INTERFACE Evaluable

METHOD evalue : Awaitable
VAR_INPUT
	value: BOOL;
	onTrueCallback: Callback;
	onFalseCallback: REFERENCE TO AwaitableError;
	message: STRING(255);
END_VAR
END_METHOD

END_INTERFACE

(* stored: Version 1.1.0.1, ProductVersion 3.1.4024.12
   Itf Evaluable: Id {5fdc8daf-5053-4b6d-a120-f929bb45a04c}
   Method evalue: Id {ba9f3a6b-fa87-4866-871a-3fd79ff26bc8} *)
